Staubli VAL3: AxisJogSpeed.pgx

public program AxisJogSpeed(num x_nSpeed, bool x_b8Axis)
begin

  //修改点动速度
  //修改1这个是比例系数

  x_nSpeed=max(0,min(100,x_nSpeed))
  if x_b8Axis

    aioSet(aAio["O4_a8JogVelo"],x_nSpeed*1)

  else
    aioSet(aAio["O4_a7JogVelo"],x_nSpeed*1)

  endIf




end
